PROGRAM MAIN
VAR
    relay : Relay;
    oven : Oven;
END_VAR

// Oven command comes from the HMI
oven(relayState:=relay._state);
relay(_command:=oven.relayCommand);

END_PROGRAM

(* stored: Version 1.1.0.1, ProductVersion 3.1.4024.4
   POU MAIN: Id {fb3609b4-3109-466e-87e3-78da51fdfb50}, SpecialFunc None *)
